KUKA KRL program: B3_Parca_Birakma.src, B3_Parca_Birakma.dat

--- B3_Parca_Birakma.src ---
&ACCESS RVP1
&REL 100
&PARAM DISKPATH = KRC:\R1\Program\Parca_Birakma
DEF  B3_Parca_Birakma ( )

   ;FOLD INI;%{PE}
   ;FOLD BASISTECH INI
   GLOBAL INTERRUPT DECL 3 WHEN $STOPMESS==TRUE DO IR_STOPM ( )
   INTERRUPT ON 3
   BAS (#INITMOV,0 )
   ;ENDFOLD (BASISTECH INI)
   ;FOLD USER INI
   ;Make your modifications here

   ;ENDFOLD (USER INI)
   ;ENDFOLD (INI)
   CONTINUE
   WAIT FOR $IN[113]==TRUE

   ; ============================================================
   ; CALCULATIONS
   ; ============================================================
   Parca_Hesaplama()
   Palet_Dom_Exp_Hesaplama()
   Pick_Point_Offs()
   B3_Palet_Hesaplama()
   Dizilim_B3 = Dizilim
   Kat_Kontrol_B3()
   ;FOLD SPTP HOME CONT Vel=100 % DEFAULT ;%{PE}
   ;FOLD Parameters ;%{h}
   ;Params IlfProvider=kukaroboter.basistech.inlineforms.movement.spline; Kuka.IsGlobalPoint=False; Kuka.PointName=HOME; Kuka.BlendingEnabled=True; Kuka.MoveDataPtpName=DEFAULT; Kuka.VelocityPtp=100; Kuka.CurrentCDSetIndex=0; Kuka.MovementParameterFieldEnabled=True; IlfCommand=SPTP
   ;ENDFOLD
   $BWDSTART = FALSE
   PDAT_ACT = PDEFAULT
   FDAT_ACT = FHOME
   BAS(#PTP_PARAMS, 100.0)
   SET_CD_PARAMS (0)
   SPTP XHOME C_SPL
   ;ENDFOLD

   ; ============================================================
   ; APPROACH PICK
   ; ============================================================
   ;FOLD SPTP Pre_Pick_Point CONT Vel=100 % PDAT2 Tool[1]:Gripper Base[0] ;%{PE}
   ;FOLD Parameters ;%{h}
   ;Params IlfProvider=kukaroboter.basistech.inlineforms.movement.spline; Kuka.IsGlobalPoint=False; Kuka.PointName=Pre_Pick_Point; Kuka.BlendingEnabled=True; Kuka.MoveDataPtpName=PDAT2; Kuka.VelocityPtp=100; Kuka.CurrentCDSetIndex=0; Kuka.MovementParameterFieldEnabled=True; IlfCommand=SPTP
   ;ENDFOLD
   $BWDSTART = FALSE
   PDAT_ACT = PPDAT2
   FDAT_ACT = FPre_Pick_Point
   BAS(#PTP_PARAMS, 100.0)
   SET_CD_PARAMS (0)
   SPTP XPre_Pick_Point C_SPL
   ;ENDFOLD

   ; ============================================================
   ; PICK ACTION
   ; ============================================================
   TRIGGER WHEN DISTANCE=0 DELAY=-0.5 DO Parca_Agirlik_Ekleme() PRIO=-1
   ;FOLD SLIN Pick_Point Vel=3 m/s CPDAT3 Tool[1]:Gripper Base[0] ;%{PE}
   ;FOLD Parameters ;%{h}
   ;Params IlfProvider=kukaroboter.basistech.inlineforms.movement.spline; Kuka.IsGlobalPoint=False; Kuka.PointName=Pick_Point; Kuka.BlendingEnabled=False; Kuka.MoveDataName=CPDAT3; Kuka.VelocityPath=3; Kuka.CurrentCDSetIndex=0; Kuka.MovementParameterFieldEnabled=True; IlfCommand=SLIN
   ;ENDFOLD
   $BWDSTART = FALSE
   LDAT_ACT = LCPDAT3
   FDAT_ACT = FPick_Point
   BAS(#CP_PARAMS, 3.0)
   SET_CD_PARAMS (0)
   ; TRIGGER: Output 189=TRUE (Gripper Open Cmd), 190=FALSE (Gripper Close Cmd)
   TRIGGER WHEN DISTANCE= 0 DELAY=0 DO $OUT[189]=TRUE
   TRIGGER WHEN DISTANCE= 0 DELAY=0 DO $OUT[190]=FALSE
   SLIN XPick_Point
   ;ENDFOLD

  CONTINUE
  WAIT FOR $IN[39]==TRUE
  CONTINUE
  $OUT[189]=FALSE
  CONTINUE
  $OUT[44]=TRUE
  CONTINUE
  $OUT[57]=TRUE


   CONTINUE
   WAIT FOR $IN[114]==TRUE
   CONTINUE
   $OUT[57]=FALSE
   CONTINUE
   $OUT[155]=FALSE



   IF (First_Start_B3==TRUE) THEN
      Bolge_3_Palet_Ort()
      First_Start_B3=FALSE
   ENDIF
   Parca_Dizilim(B3_ParcaSirasi,B3_ParcaKatSayisi,3)
   B3_Parca_Konum_Hesaplama()

   ; ============================================================
   ; TRANSPORT
   ; ============================================================
   ;FOLD SPTP B5_PARCA_BIRAKMA CONT Vel=100 % PDAT4 Tool[1]:Gripper Base[0] ;%{PE}
   ;FOLD Parameters ;%{h}
   ;Params IlfProvider=kukaroboter.basistech.inlineforms.movement.spline; Kuka.IsGlobalPoint=False; Kuka.PointName=B5_PARCA_BIRAKMA; Kuka.BlendingEnabled=True; Kuka.MoveDataPtpName=PDAT4; Kuka.VelocityPtp=100; Kuka.CurrentCDSetIndex=0; Kuka.MovementParameterFieldEnabled=True; IlfCommand=SPTP
   ;ENDFOLD
   $BWDSTART = FALSE
   PDAT_ACT = PPDAT4
   FDAT_ACT = FB5_PARCA_BIRAKMA
   BAS(#PTP_PARAMS, 100.0)
   SET_CD_PARAMS (0)
   SPTP XB5_PARCA_BIRAKMA C_SPL
   ;ENDFOLD


   ; ============================================================
   ; APPROACH PLACE
   ; ============================================================
   ;FOLD SPTP B3_ARA_NOKT CONT Vel=100 % PDAT14 Tool[1]:Gripper Base[3]:BOLGE_3 ;%{PE}
   ;FOLD Parameters ;%{h}
   ;Params IlfProvider=kukaroboter.basistech.inlineforms.movement.spline; Kuka.IsGlobalPoint=False; Kuka.PointName=B3_ARA_NOKT; Kuka.BlendingEnabled=True; Kuka.MoveDataPtpName=PDAT14; Kuka.VelocityPtp=100; Kuka.CurrentCDSetIndex=0; Kuka.MovementParameterFieldEnabled=True; IlfCommand=SPTP
   ;ENDFOLD
   $BWDSTART = FALSE
   PDAT_ACT = PPDAT14
   FDAT_ACT = FB3_ARA_NOKT
   BAS(#PTP_PARAMS, 100.0)
   SET_CD_PARAMS (0)
   SPTP XB3_ARA_NOKT C_SPL
   ;ENDFOLD
;FOLD SPTP B3_PRE_PARCA_BIRAKMA CONT Vel=100 % PDAT20 Tool[1]:Gripper Base[3]:BOLGE_3 ;%{PE}
;FOLD Parameters ;%{h}
;Params IlfProvider=kukaroboter.basistech.inlineforms.movement.spline; Kuka.IsGlobalPoint=False; Kuka.PointName=B3_PRE_PARCA_BIRAKMA; Kuka.BlendingEnabled=True; Kuka.MoveDataPtpName=PDAT20; Kuka.VelocityPtp=100; Kuka.VelocityFieldEnabled=True; Kuka.ColDetectFieldEnabled=True; Kuka.CurrentCDSetIndex=0; Kuka.MovementParameterFieldEnabled=True; IlfCommand=SPTP
;ENDFOLD
SPTP XB3_PRE_PARCA_BIRAKMA WITH $VEL_AXIS[1] = SVEL_JOINT(100.0), $TOOL = STOOL2(FB3_PRE_PARCA_BIRAKMA), $BASE = SBASE(FB3_PRE_PARCA_BIRAKMA.BASE_NO), $IPO_MODE = SIPO_MODE(FB3_PRE_PARCA_BIRAKMA.IPO_FRAME), $LOAD = SLOAD(FB3_PRE_PARCA_BIRAKMA.TOOL_NO), $ACC_AXIS[1] = SACC_JOINT(PPDAT20), $APO = SAPO_PTP(PPDAT20), $GEAR_JERK[1] = SGEAR_JERK(PPDAT20), $COLLMON_TOL_PRO[1] = USE_CM_PRO_VALUES(0) C_Spl
;ENDFOLD

   ; ============================================================
   ; PLACE ACTION
   ; ============================================================
   ;FOLD SLIN B3_PARCA_BIRAKMA Vel=3.0 m/s CPDAT9 Tool[1]:Gripper Base[3]:BOLGE_3 ;%{PE}
   ;FOLD Parameters ;%{h}
   ;Params IlfProvider=kukaroboter.basistech.inlineforms.movement.spline; Kuka.IsGlobalPoint=False; Kuka.PointName=B3_PARCA_BIRAKMA; Kuka.BlendingEnabled=False; Kuka.MoveDataName=CPDAT9; Kuka.VelocityPath=3.0; Kuka.CurrentCDSetIndex=0; Kuka.MovementParameterFieldEnabled=True; IlfCommand=SLIN
   ;ENDFOLD
   $BWDSTART = FALSE
   LDAT_ACT = LCPDAT9
   FDAT_ACT = FB3_PARCA_BIRAKMA
   BAS(#CP_PARAMS, 3.0)
   SET_CD_PARAMS (0)
   ;TRIGGER WHEN DISTANCE=0 DELAY=0 DO $OUT[190]=TRUE
   ;TRIGGER WHEN DISTANCE=0 DELAY=0 DO $OUT[189]=FALSE
   SLIN XB3_PARCA_BIRAKMA
   ;ENDFOLD

   $OUT[190]=TRUE
   $OUT[189]=FALSE
   CONTINUE
   WAIT FOR $IN[40]==TRUE
   CONTINUE
   $OUT[44]=FALSE

   ; ============================================================
   ; DEPART PLACE
   ; ============================================================
   ;FOLD SLIN B3_PRE_PARCA_BIRAKMA CONT Vel=3.0 m/s CPDAT1 Tool[1]:Gripper Base[3]:BOLGE_3 ;%{PE}
   ;FOLD Parameters ;%{h}
   ;Params IlfProvider=kukaroboter.basistech.inlineforms.movement.spline; Kuka.IsGlobalPoint=False; Kuka.PointName=B3_PRE_PARCA_BIRAKMA; Kuka.BlendingEnabled=True; Kuka.MoveDataName=CPDAT1; Kuka.VelocityPath=3.0; Kuka.CurrentCDSetIndex=0; Kuka.MovementParameterFieldEnabled=True; IlfCommand=SLIN
   ;ENDFOLD
   $BWDSTART = FALSE
   LDAT_ACT = LCPDAT1
   FDAT_ACT = FB3_PRE_PARCA_BIRAKMA
   BAS(#CP_PARAMS, 3.0)
   SET_CD_PARAMS (0)
   TRIGGER WHEN DISTANCE=0 DELAY=-0.3 DO $OUT[58]=TRUE
   SLIN XB3_PRE_PARCA_BIRAKMA C_SPL
   ;ENDFOLD

   ;FOLD SPTP B3_ARA_NOKT CONT Vel=100 % PDAT17 Tool[1]:Gripper Base[3]:BOLGE_3 ;%{PE}
   ;FOLD Parameters ;%{h}
   ;Params IlfProvider=kukaroboter.basistech.inlineforms.movement.spline; Kuka.IsGlobalPoint=False; Kuka.PointName=B3_ARA_NOKT; Kuka.BlendingEnabled=True; Kuka.MoveDataPtpName=PDAT17; Kuka.VelocityPtp=100; Kuka.CurrentCDSetIndex=0; Kuka.MovementParameterFieldEnabled=True; IlfCommand=SPTP
   ;ENDFOLD
   $BWDSTART = FALSE
   PDAT_ACT = PPDAT17
   FDAT_ACT = FB3_ARA_NOKT
   BAS(#PTP_PARAMS, 100.0)
   SET_CD_PARAMS (0)
   TRIGGER WHEN DISTANCE=0 DELAY=-0.3 DO $OUT[190]=FALSE
   SPTP XB3_ARA_NOKT C_SPL
   ;ENDFOLD

   ;FOLD SPTP pre_home CONT Vel=100 % PDAT18 Tool[1]:Gripper Base[0] ;%{PE}
   ;FOLD Parameters ;%{h}
   ;Params IlfProvider=kukaroboter.basistech.inlineforms.movement.spline; Kuka.IsGlobalPoint=False; Kuka.PointName=pre_home; Kuka.BlendingEnabled=True; Kuka.MoveDataPtpName=PDAT18; Kuka.VelocityPtp=100; Kuka.CurrentCDSetIndex=0; Kuka.MovementParameterFieldEnabled=True; IlfCommand=SPTP
   ;ENDFOLD
   $BWDSTART = FALSE
   PDAT_ACT = PPDAT18
   FDAT_ACT = Fpre_home
   BAS(#PTP_PARAMS, 100.0)
   SET_CD_PARAMS (0)
   SPTP Xpre_home C_SPL
   ;ENDFOLD
   ;FOLD SPTP HOME Vel=100 % DEFAULT ;%{PE}
   ;FOLD Parameters ;%{h}
   ;Params IlfProvider=kukaroboter.basistech.inlineforms.movement.spline; Kuka.IsGlobalPoint=False; Kuka.PointName=HOME; Kuka.BlendingEnabled=False; Kuka.MoveDataPtpName=DEFAULT; Kuka.VelocityPtp=100; Kuka.CurrentCDSetIndex=0; Kuka.MovementParameterFieldEnabled=True; IlfCommand=SPTP
   ;ENDFOLD
   $BWDSTART = FALSE
   PDAT_ACT = PDEFAULT
   FDAT_ACT = FHOME
   BAS(#PTP_PARAMS, 100.0)
   SET_CD_PARAMS (0)
   TRIGGER WHEN DISTANCE=0 DELAY=-0.3 DO $OUT[58]=FALSE
   TRIGGER WHEN DISTANCE=0 DELAY=-0.3 DO $OUT[155]=TRUE
   SPTP XHOME
   ;ENDFOLD
   B3_Kat_Hesaplama()

END

--- B3_Parca_Birakma.dat ---
&ACCESS RVP1
&REL 101
&PARAM DISKPATH = KRC:\R1\Program\Parca_Birakma
DEFDAT  B3_PARCA_BIRAKMA
;FOLD EXTERNAL DECLARATIONS;%{PE}%MKUKATPBASIS,%CEXT,%VCOMMON,%P
;FOLD BASISTECH EXT;%{PE}%MKUKATPBASIS,%CEXT,%VEXT,%P
EXT  BAS (BAS_COMMAND  :IN,REAL  :IN )
DECL INT SUCCESS
;ENDFOLD (BASISTECH EXT)
;FOLD USER EXT;%{E}%MKUKATPUSER,%CEXT,%VEXT,%P
;Make your modifications here

;ENDFOLD (USER EXT)
;ENDFOLD (EXTERNAL DECLARATIONS)
DECL FDAT FPre_Pick_Point={TOOL_NO 1,BASE_NO 0,IPO_FRAME #BASE,POINT2[] " "}
DECL FDAT FPick_Point={TOOL_NO 1,BASE_NO 0,IPO_FRAME #BASE,POINT2[] " "}
DECL FDAT FB3_PARCA_BIRAKMA={TOOL_NO 1,BASE_NO 3,IPO_FRAME #BASE,POINT2[] " "}
DECL PDAT PPDAT1={VEL 100.000,ACC 100.000,APO_DIST 500.000,APO_MODE #CDIS,GEAR_JERK 100.000,EXAX_IGN 0}
DECL MODULEPARAM_T LAST_TP_PARAMS={PARAMS[] "Kuka.PointName=B3_PRE_PARCA_BIRAKMA; Kuka.FrameData.base_no=3; Kuka.FrameData.tool_no=1; Kuka.FrameData.ipo_frame=#BASE; Kuka.FrameData.point2=; Kuka.isglobalpoint=False; Kuka.MoveDataPtpName=PDAT20; Kuka.MovementDataPdat.apo_mode=#CDIS; Kuka.MovementDataPdat.apo_dist=500; Kuka.MovementData.vel=100; Kuka.MovementData.acc=100; Kuka.MovementData.exax_ign=0; Kuka.VelocityPtp=100; Kuka.BlendingEnabled=True; Kuka.APXEnabled=False; Kuka.CurrentCDSetIndex=0; Kuka.VelocityFieldEnabled=True; Kuka.ColDetectFieldEnabled=True; Kuka.MovementParameterFieldEnabled=True; Kuka.IsAngleEnabled=False; Kuka.MoveDataName=CPDAT13; Kuka.MovementData.cb={AUX_PT {ORI #CONSIDER,E1 #CONSIDER,E2 #CONSIDER,E3 #CONSIDER,E4 #CONSIDER,E5 #CONSIDER,E6 #CONSIDER},TARGET_PT {ORI #INTERPOLATE,E1 #INTERPOLATE,E2 #INTERPOLATE,E3 #INTERPOLATE,E4 #INTERPOLATE,E5 #INTERPOLATE,E6 #INTERPOLATE}}; Kuka.MovementData.apo_fac=50; Kuka.MovementData.apo_dist=500; Kuka.MovementData.axis_acc=100; Kuka.MovementData.axis_vel=100; Kuka.MovementData.circ_typ=#BASE; Kuka.MovementData.jerk_fac=50; Kuka.MovementData.ori_typ=#VAR; Kuka.VelocityPath=1.3   "}

DECL FDAT FB3_ARA_NOKT={TOOL_NO 1,BASE_NO 3,IPO_FRAME #BASE,POINT2[] " "}
DECL PDAT PPDAT2={VEL 100.000,ACC 100.000,APO_DIST 500.000,APO_MODE #CDIS,GEAR_JERK 100.000,EXAX_IGN 0}

DECL FDAT FB3_PRE_PARCA_BIRAKMA={TOOL_NO 1,BASE_NO 3,IPO_FRAME #BASE,POINT2[] " "}
DECL PDAT PPDAT3={VEL 100.000,ACC 100.000,APO_DIST 500.000,APO_MODE #CDIS,GEAR_JERK 100.000,EXAX_IGN 0}
DECL LDAT LCPDAT1={VEL 1.30000,ACC 100.000,APO_DIST 500.000,APO_FAC 50.0000,AXIS_VEL 100.000,AXIS_ACC 100.000,ORI_TYP #VAR,CIRC_TYP #BASE,JERK_FAC 50.0000,GEAR_JERK 100.000,EXAX_IGN 0,CB {AUX_PT {ORI #CONSIDER,E1 #CONSIDER,E2 #CONSIDER,E3 #CONSIDER,E4 #CONSIDER,E5 #CONSIDER,E6 #CONSIDER},TARGET_PT {ORI #INTERPOLATE,E1 #INTERPOLATE,E2 #INTERPOLATE,E3 #INTERPOLATE,E4 #INTERPOLATE,E5 #INTERPOLATE,E6 #INTERPOLATE}}}
DECL LDAT LCPDAT2={VEL 2.00000,ACC 100.000,APO_DIST 500.000,APO_FAC 50.0000,AXIS_VEL 100.000,AXIS_ACC 100.000,ORI_TYP #VAR,CIRC_TYP #BASE,JERK_FAC 50.0000,GEAR_JERK 100.000,EXAX_IGN 0,CB {AUX_PT {ORI #CONSIDER,E1 #CONSIDER,E2 #CONSIDER,E3 #CONSIDER,E4 #CONSIDER,E5 #CONSIDER,E6 #CONSIDER},TARGET_PT {ORI #INTERPOLATE,E1 #INTERPOLATE,E2 #INTERPOLATE,E3 #INTERPOLATE,E4 #INTERPOLATE,E5 #INTERPOLATE,E6 #INTERPOLATE}}}

DECL FDAT FB5_PARCA_BIRAKMA={TOOL_NO 1,BASE_NO 0,IPO_FRAME #BASE,POINT2[] " "}
DECL PDAT PPDAT4={VEL 100.000,ACC 100.000,APO_DIST 500.000,APO_MODE #CDIS,GEAR_JERK 100.000,EXAX_IGN 0}
DECL LDAT LCPDAT3={VEL 1.50000,ACC 100.000,APO_DIST 500.000,APO_FAC 50.0000,AXIS_VEL 100.000,AXIS_ACC 100.000,ORI_TYP #VAR,CIRC_TYP #BASE,JERK_FAC 50.0000,GEAR_JERK 100.000,EXAX_IGN 0,CB {AUX_PT {ORI #CONSIDER,E1 #CONSIDER,E2 #CONSIDER,E3 #CONSIDER,E4 #CONSIDER,E5 #CONSIDER,E6 #CONSIDER},TARGET_PT {ORI #INTERPOLATE,E1 #INTERPOLATE,E2 #INTERPOLATE,E3 #INTERPOLATE,E4 #INTERPOLATE,E5 #INTERPOLATE,E6 #INTERPOLATE}}}
DECL LDAT LCPDAT4={VEL 3.00000,ACC 100.000,APO_DIST 500.000,APO_FAC 50.0000,AXIS_VEL 100.000,AXIS_ACC 100.000,ORI_TYP #VAR,CIRC_TYP #BASE,JERK_FAC 50.0000,GEAR_JERK 100.000,EXAX_IGN 0,CB {AUX_PT {ORI #CONSIDER,E1 #CONSIDER,E2 #CONSIDER,E3 #CONSIDER,E4 #CONSIDER,E5 #CONSIDER,E6 #CONSIDER},TARGET_PT {ORI #INTERPOLATE,E1 #INTERPOLATE,E2 #INTERPOLATE,E3 #INTERPOLATE,E4 #INTERPOLATE,E5 #INTERPOLATE,E6 #INTERPOLATE}}}
DECL PDAT PPDAT5={VEL 100.000,ACC 100.000,APO_DIST 500.000,APO_MODE #CDIS,GEAR_JERK 100.000,EXAX_IGN 0}
DECL LDAT LCPDAT5={VEL 3.00000,ACC 100.000,APO_DIST 500.000,APO_FAC 50.0000,AXIS_VEL 100.000,AXIS_ACC 100.000,ORI_TYP #VAR,CIRC_TYP #BASE,JERK_FAC 50.0000,GEAR_JERK 100.000,EXAX_IGN 0,CB {AUX_PT {ORI #CONSIDER,E1 #CONSIDER,E2 #CONSIDER,E3 #CONSIDER,E4 #CONSIDER,E5 #CONSIDER,E6 #CONSIDER},TARGET_PT {ORI #INTERPOLATE,E1 #INTERPOLATE,E2 #INTERPOLATE,E3 #INTERPOLATE,E4 #INTERPOLATE,E5 #INTERPOLATE,E6 #INTERPOLATE}}}
DECL PDAT PPDAT6={VEL 100.000,ACC 100.000,APO_DIST 500.000,APO_MODE #CDIS,GEAR_JERK 100.000,EXAX_IGN 0}

DECL FDAT Fb3_arankta={TOOL_NO 1,BASE_NO 0,IPO_FRAME #BASE,POINT2[] " "}
DECL LDAT LCPDAT6={VEL 3.00000,ACC 100.000,APO_DIST 500.000,APO_FAC 50.0000,AXIS_VEL 100.000,AXIS_ACC 100.000,ORI_TYP #VAR,CIRC_TYP #BASE,JERK_FAC 50.0000,GEAR_JERK 100.000,EXAX_IGN 0,CB {AUX_PT {ORI #CONSIDER,E1 #CONSIDER,E2 #CONSIDER,E3 #CONSIDER,E4 #CONSIDER,E5 #CONSIDER,E6 #CONSIDER},TARGET_PT {ORI #INTERPOLATE,E1 #INTERPOLATE,E2 #INTERPOLATE,E3 #INTERPOLATE,E4 #INTERPOLATE,E5 #INTERPOLATE,E6 #INTERPOLATE}}}
DECL LDAT LCPDAT7={VEL 3.00000,ACC 100.000,APO_DIST 500.000,APO_FAC 50.0000,AXIS_VEL 100.000,AXIS_ACC 100.000,ORI_TYP #VAR,CIRC_TYP #BASE,JERK_FAC 50.0000,GEAR_JERK 100.000,EXAX_IGN 0,CB {AUX_PT {ORI #CONSIDER,E1 #CONSIDER,E2 #CONSIDER,E3 #CONSIDER,E4 #CONSIDER,E5 #CONSIDER,E6 #CONSIDER},TARGET_PT {ORI #INTERPOLATE,E1 #INTERPOLATE,E2 #INTERPOLATE,E3 #INTERPOLATE,E4 #INTERPOLATE,E5 #INTERPOLATE,E6 #INTERPOLATE}}}
DECL PDAT PPDAT7={VEL 100.000,ACC 100.000,APO_DIST 500.000,APO_MODE #CDIS,GEAR_JERK 100.000,EXAX_IGN 0}
DECL LDAT LCPDAT8={VEL 3.00000,ACC 100.000,APO_DIST 500.000,APO_FAC 50.0000,AXIS_VEL 100.000,AXIS_ACC 100.000,ORI_TYP #VAR,CIRC_TYP #BASE,JERK_FAC 50.0000,GEAR_JERK 100.000,EXAX_IGN 0,CB {AUX_PT {ORI #CONSIDER,E1 #CONSIDER,E2 #CONSIDER,E3 #CONSIDER,E4 #CONSIDER,E5 #CONSIDER,E6 #CONSIDER},TARGET_PT {ORI #INTERPOLATE,E1 #INTERPOLATE,E2 #INTERPOLATE,E3 #INTERPOLATE,E4 #INTERPOLATE,E5 #INTERPOLATE,E6 #INTERPOLATE}}}
DECL PDAT PPDAT8={VEL 100.000,ACC 100.000,APO_DIST 500.000,APO_MODE #CDIS,GEAR_JERK 100.000,EXAX_IGN 0}
DECL PDAT PPDAT9={VEL 100.000,ACC 100.000,APO_DIST 500.000,APO_MODE #CDIS,GEAR_JERK 100.000,EXAX_IGN 0}
DECL LDAT LCPDAT9={VEL 3.00000,ACC 100.000,APO_DIST 500.000,APO_FAC 50.0000,AXIS_VEL 100.000,AXIS_ACC 100.000,ORI_TYP #VAR,CIRC_TYP #BASE,JERK_FAC 50.0000,GEAR_JERK 100.000,EXAX_IGN 0,CB {AUX_PT {ORI #CONSIDER,E1 #CONSIDER,E2 #CONSIDER,E3 #CONSIDER,E4 #CONSIDER,E5 #CONSIDER,E6 #CONSIDER},TARGET_PT {ORI #INTERPOLATE,E1 #INTERPOLATE,E2 #INTERPOLATE,E3 #INTERPOLATE,E4 #INTERPOLATE,E5 #INTERPOLATE,E6 #INTERPOLATE}}}
DECL LDAT LCPDAT10={VEL 3.00000,ACC 100.000,APO_DIST 500.000,APO_FAC 50.0000,AXIS_VEL 100.000,AXIS_ACC 100.000,ORI_TYP #VAR,CIRC_TYP #BASE,JERK_FAC 50.0000,GEAR_JERK 100.000,EXAX_IGN 0,CB {AUX_PT {ORI #CONSIDER,E1 #CONSIDER,E2 #CONSIDER,E3 #CONSIDER,E4 #CONSIDER,E5 #CONSIDER,E6 #CONSIDER},TARGET_PT {ORI #INTERPOLATE,E1 #INTERPOLATE,E2 #INTERPOLATE,E3 #INTERPOLATE,E4 #INTERPOLATE,E5 #INTERPOLATE,E6 #INTERPOLATE}}}
DECL PDAT PPDAT10={VEL 100.000,ACC 100.000,APO_DIST 500.000,APO_MODE #CDIS,GEAR_JERK 100.000,EXAX_IGN 0}
DECL LDAT LCPDAT11={VEL 3.00000,ACC 100.000,APO_DIST 500.000,APO_FAC 50.0000,AXIS_VEL 100.000,AXIS_ACC 100.000,ORI_TYP #VAR,CIRC_TYP #BASE,JERK_FAC 50.0000,GEAR_JERK 100.000,EXAX_IGN 0,CB {AUX_PT {ORI #CONSIDER,E1 #CONSIDER,E2 #CONSIDER,E3 #CONSIDER,E4 #CONSIDER,E5 #CONSIDER,E6 #CONSIDER},TARGET_PT {ORI #INTERPOLATE,E1 #INTERPOLATE,E2 #INTERPOLATE,E3 #INTERPOLATE,E4 #INTERPOLATE,E5 #INTERPOLATE,E6 #INTERPOLATE}}}
DECL PDAT PPDAT11={VEL 100.000,ACC 100.000,APO_DIST 500.000,APO_MODE #CDIS,GEAR_JERK 100.000,EXAX_IGN 0}
DECL LDAT LCPDAT12={VEL 1.30000,ACC 100.000,APO_DIST 500.000,APO_FAC 50.0000,AXIS_VEL 100.000,AXIS_ACC 100.000,ORI_TYP #VAR,CIRC_TYP #BASE,JERK_FAC 50.0000,GEAR_JERK 100.000,EXAX_IGN 0,CB {AUX_PT {ORI #CONSIDER,E1 #CONSIDER,E2 #CONSIDER,E3 #CONSIDER,E4 #CONSIDER,E5 #CONSIDER,E6 #CONSIDER},TARGET_PT {ORI #INTERPOLATE,E1 #INTERPOLATE,E2 #INTERPOLATE,E3 #INTERPOLATE,E4 #INTERPOLATE,E5 #INTERPOLATE,E6 #INTERPOLATE}}}
DECL E6POS XB6_PRE_PARCA_BIRAKMA={X -32.0079269,Y -487.505157,Z 223.679276,A 179.999741,B -3.73135665E-14,C -6.13378532E-12,S 2,T 32,E1 0.0,E2 0.0,E3 0.0,E4 0.0,E5 0.0,E6 0.0}
DECL FDAT FB6_PRE_PARCA_BIRAKMA={TOOL_NO 1,BASE_NO 3,IPO_FRAME #BASE,POINT2[] " "}
DECL PDAT PPDAT12={VEL 100.000,ACC 100.000,APO_DIST 500.000,APO_MODE #CDIS,GEAR_JERK 100.000,EXAX_IGN 0}
DECL PDAT PPDAT13={VEL 100.000,ACC 100.000,APO_DIST 500.000,APO_MODE #CDIS,GEAR_JERK 100.000,EXAX_IGN 0}
DECL PDAT PPDAT14={VEL 100.000,ACC 100.000,APO_DIST 500.000,APO_MODE #CDIS,GEAR_JERK 100.000,EXAX_IGN 0}
DECL PDAT PPDAT15={VEL 100.000,ACC 100.000,APO_DIST 500.000,APO_MODE #CDIS,GEAR_JERK 100.000,EXAX_IGN 0}
DECL LDAT LCPDAT13={VEL 1.30000,ACC 100.000,APO_DIST 500.000,APO_FAC 50.0000,AXIS_VEL 100.000,AXIS_ACC 100.000,ORI_TYP #VAR,CIRC_TYP #BASE,JERK_FAC 50.0000,GEAR_JERK 100.000,EXAX_IGN 0,CB {AUX_PT {ORI #CONSIDER,E1 #CONSIDER,E2 #CONSIDER,E3 #CONSIDER,E4 #CONSIDER,E5 #CONSIDER,E6 #CONSIDER},TARGET_PT {ORI #INTERPOLATE,E1 #INTERPOLATE,E2 #INTERPOLATE,E3 #INTERPOLATE,E4 #INTERPOLATE,E5 #INTERPOLATE,E6 #INTERPOLATE}}}
DECL E6POS XB4_ARA_NOKT={X -50.4699402,Y -110.191841,Z 1594.13843,A 179.367599,B -1.18816979E-12,C -7.73512157E-12,S 2,T 10,E1 0.0,E2 0.0,E3 0.0,E4 0.0,E5 0.0,E6 0.0}
DECL FDAT FB4_ARA_NOKT={TOOL_NO 1,BASE_NO 3,IPO_FRAME #BASE,POINT2[] " "}
DECL PDAT PPDAT16={VEL 100.000,ACC 100.000,APO_DIST 500.000,APO_MODE #CDIS,GEAR_JERK 100.000,EXAX_IGN 0}
DECL PDAT PPDAT17={VEL 100.000,ACC 100.000,APO_DIST 500.000,APO_MODE #CDIS,GEAR_JERK 100.000,EXAX_IGN 0}
DECL E6POS Xpre_home={X 1753.58252,Y -5.82854223,Z 876.082520,A 0.00291636912,B 1.88846595E-12,C -3.02852578E-12,S 2,T 2,E1 0.0,E2 0.0,E3 0.0,E4 0.0,E5 0.0,E6 0.0}
DECL FDAT Fpre_home={TOOL_NO 1,BASE_NO 0,IPO_FRAME #BASE,POINT2[] " "}
DECL PDAT PPDAT18={VEL 100.000,ACC 100.000,APO_DIST 500.000,APO_MODE #CDIS,GEAR_JERK 100.000,EXAX_IGN 0}
DECL FDAT FPre_Pick_Point_1={TOOL_NO 1,BASE_NO 0,IPO_FRAME #BASE,POINT2[] " "}
DECL PDAT PPDAT19={VEL 100.000,ACC 100.000,APO_DIST 581.000,APO_MODE #CDIS,GEAR_JERK 100.000,EXAX_IGN 0}
DECL PDAT PPDAT20={VEL 100.000,ACC 100.000,APO_DIST 500.000,APO_MODE #CDIS,GEAR_JERK 100.000,EXAX_IGN 0}
ENDDAT
